// TIA Portal V20 export
VAR_GLOBAL   // PLC tag table "Circuit Breaker"
END_VAR
